(* CODESYS project Test FB.project

Project tree, tasks and I/O mapping:
  Device : CODESYS Control Win V3, 3S - Smart Software Solutions GmbH, version 3.5.15.30
    application Application
      libraries: Standard, * (System)
      task MainTask (cyclic, interval t#20ms, priority 1) calls PLC_PRG
      task VISU_TASK (cyclic, interval 100 ms, priority 31) calls VisuElems.Visu_Prg
      program PLC_PRG [FBD]
      visualisation Visualization
  text list GlobalTextList
*)

// Device/Application/PLC_PRG
PROGRAM PLC_PRG
VAR
	CTU_0: CTU;
	Contact1 : BOOL;
	PV1 : WORD := 3;
	Value : WORD;
	Coil1 : BOOL;
	Reset : BOOL;
END_VAR

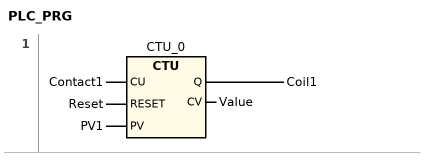
// NETWORK 1
CTU_0(CU := Contact1, RESET := Reset, PV := PV1, CV => Value); // CTU
Coil1 := CTU_0.Q;

END_PROGRAM

// Device/Application/Visualization
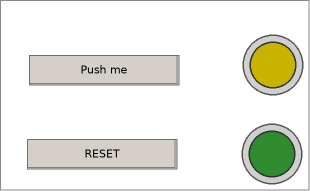
VISUALIZATION Visualization  // 310x191
    Lamp1 (238,30 70x70), variable: PLC_PRG.Coil1, style: Lamp-Lamp1-Yellow
    Button (29,55 150x30), "Push me"
        tap PLC_PRG.Contact1
    Button (27,139 150x30), "RESET"
        tap PLC_PRG.Reset
    Lamp1 (237,119 70x70), variable: PLC_PRG.CTU_0.Q, style: Lamp-Lamp1-Green
END_VISUALIZATION
